{attribute 'qualified_only'}
{attribute 'strict'}

//-----------------------------------------------------------------------------------------
//
//                  				ENUM_Jog_Mode
//
//						Enumération des Modes des Axes en Jog			
//-----------------------------------------------------------------------------------------
//
//Auteur: G.GOETZ
//Création: 19.01.2026
//Dernière modification : 19.01.2026 (G.GOETZ)
//       			
//-----------------------------------------------------------------------------------------
//
//     							Liste des modifications  	
//
// 19.01.2026 (G.GOETZ) -> Création		
//-----------------------------------------------------------------------------------------

TYPE ENUM_Jog_Mode :
(
	None := 0 , // Unknow Mode
	Inching := 1 , // Inching Mode = Incremental
	Continous := 2 // Continous Mode = Jog
);
END_TYPE

(* stored: Version 1.1.0.1, ProductVersion 3.1.4026.17
   DUT ENUM_Jog_Mode: Id {bae63465-674a-4efe-8a71-a07b563a212d} *)
